TYPE E_ValveStatus :
(
	OK,
    SHORT_CIRCUIT,
    OPEN_CIRCUIT,
    MANUAL_OVERRIDE,
    UNKNOWN_FAULT
	//OPENED_OK,  	//IF position sensor available
	//CLOSED_OK		//IF position sensor available
);
END_TYPE

(* stored: Version 1.1.0.1, ProductVersion 3.1.4024.15
   DUT E_ValveStatus: Id {a264725b-6341-48d1-95b9-c99dcd888f78} *)
